FUNCTION_BLOCK HOME_RUN_SEQ
VAR_IN_OUT
	xExecute:		BOOL;
END_VAR
VAR_OUTPUT
	xDone:			BOOL;
END_VAR
VAR
	tpReset:			TP;
	rtDone:				R_TRIG;
	rtExecute:			R_TRIG;
	ftTimePulse:		F_TRIG;
	tpTimePulse:		TP;
	lrTargetPos:		LREAL;
	xTransCondition:	BOOL;	
	xTransRelease:		BOOL;
	SFCInit:			BOOL;
	SFCReset:			BOOL;	
	SFCError:			BOOL;
END_VAR

rtDone(CLK:=xDone);
IF rtDone.Q THEN
	xTransRelease:=FALSE;	
	SFCReset:=TRUE;
END_IF

rtExecute(CLK:=xExecute);
IF rtExecute.Q THEN
	xTransRelease:=TRUE;
	SFCReset:=FALSE;
END_IF

IF xExecute THEN
	aSEQ_ACT();
END_IF

tpReset(IN:=SFCError, PT:=T#250MS);
SFCReset:= tpReset.Q;

ACTION ACK_DONE_AXIS_active:
IF G_sAxisDone.X OR G_sAxisDone.Y OR G_sAxisDone.Z OR G_sAxisDone.c THEN
	G_sAckAxisDone.X:=TRUE;
	G_sAckAxisDone.Y:=TRUE;
	G_sAckAxisDone.Z:=TRUE;
	G_sAckAxisDone.C:=TRUE;
ELSE
	G_sAckAxisDone.X:=FALSE;
	G_sAckAxisDone.Y:=FALSE;
	G_sAckAxisDone.Z:=FALSE;
	G_sAckAxisDone.C:=FALSE;
END_IF

xTransCondition:= NOT G_sAckAxisDone.X AND NOT G_sAckAxisDone.Y AND NOT G_sAckAxisDone.Z AND NOT G_sAckAxisDone.C;
END_ACTION

ACTION aSEQ_ACT:
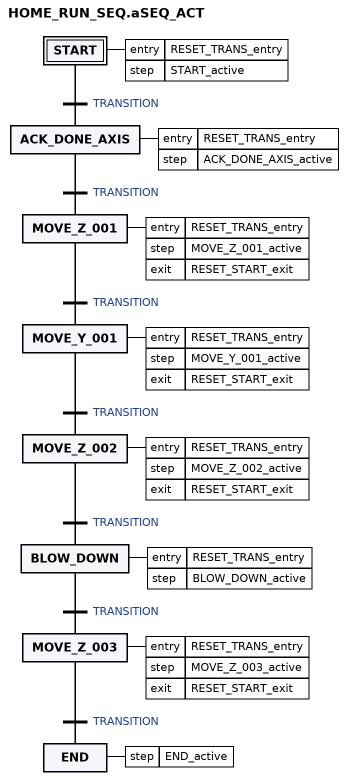
INITIAL_STEP START:
    RESET_TRANS_entry(P1);  // entry action
    START_active(N);  // step action
END_STEP
TRANSITION FROM START TO ACK_DONE_AXIS
    := TRANSITION;
END_TRANSITION
STEP ACK_DONE_AXIS:
    RESET_TRANS_entry(P1);  // entry action
    ACK_DONE_AXIS_active(N);  // step action
END_STEP
TRANSITION FROM ACK_DONE_AXIS TO MOVE_Z_001
    := TRANSITION;
END_TRANSITION
STEP MOVE_Z_001:
    RESET_TRANS_entry(P1);  // entry action
    MOVE_Z_001_active(N);  // step action
    RESET_START_exit(P0);  // exit action
END_STEP
TRANSITION FROM MOVE_Z_001 TO MOVE_Y_001
    := TRANSITION;
END_TRANSITION
STEP MOVE_Y_001:
    RESET_TRANS_entry(P1);  // entry action
    MOVE_Y_001_active(N);  // step action
    RESET_START_exit(P0);  // exit action
END_STEP
TRANSITION FROM MOVE_Y_001 TO MOVE_Z_002
    := TRANSITION;
END_TRANSITION
STEP MOVE_Z_002:
    RESET_TRANS_entry(P1);  // entry action
    MOVE_Z_002_active(N);  // step action
    RESET_START_exit(P0);  // exit action
END_STEP
TRANSITION FROM MOVE_Z_002 TO BLOW_DOWN
    := TRANSITION;
END_TRANSITION
STEP BLOW_DOWN:
    RESET_TRANS_entry(P1);  // entry action
    BLOW_DOWN_active(N);  // step action
END_STEP
TRANSITION FROM BLOW_DOWN TO MOVE_Z_003
    := TRANSITION;
END_TRANSITION
STEP MOVE_Z_003:
    RESET_TRANS_entry(P1);  // entry action
    MOVE_Z_003_active(N);  // step action
    RESET_START_exit(P0);  // exit action
END_STEP
TRANSITION FROM MOVE_Z_003 TO END
    := TRANSITION;
END_TRANSITION
STEP END:
    END_active(N);  // step action
END_STEP
END_ACTION

ACTION BLOW_DOWN_active:
tpTimePulse(IN:=NOT tpTimePulse.Q, PT:=T#3000MS);
ftTimePulse(CLK:=tpTimePulse.Q);
xTransCondition:= ftTimePulse.Q;
END_ACTION

ACTION END_active:
xDone:=TRUE;
xTransCondition:=FALSE;
END_ACTION

ACTION MOVE_Y_001_active:
G_sTargetPosition.Y:= G_asIndividualAxisPositions[CE_AXIS_Y].Positions[1].Target;
G_sStartToPos.Y:= TRUE;

xTransCondition:= G_sAxisDone.Y;
END_ACTION

ACTION MOVE_Z_001_active:
G_sTargetPosition.Z:= G_asIndividualAxisPositions[CE_AXIS_Z].Positions[1].Target;
G_sStartToPos.Z:= TRUE;

xTransCondition:= G_sAxisDone.Z;
END_ACTION

ACTION MOVE_Z_002_active:
G_sTargetPosition.Z:= G_asIndividualAxisPositions[CE_AXIS_Z].Positions[2].Target;
G_sStartToPos.Z:= TRUE;

xTransCondition:= G_sAxisDone.Z;
END_ACTION

ACTION MOVE_Z_003_active:
G_sTargetPosition.Z:= G_asIndividualAxisPositions[CE_AXIS_Z].Positions[1].Target;
G_sStartToPos.Z:= TRUE;

xTransCondition:= G_sAxisDone.Z;
END_ACTION

ACTION RESET_START_exit:
IF G_sAxisDone.X OR G_sAxisDone.Y OR G_sAxisDone.Z OR G_sAxisDone.c THEN
	G_sAckAxisDone.X:=TRUE;
	G_sAckAxisDone.Y:=TRUE;
	G_sAckAxisDone.Z:=TRUE;
	G_sAckAxisDone.C:=TRUE;
ELSE
	G_sAckAxisDone.X:=FALSE;
	G_sAckAxisDone.Y:=FALSE;
	G_sAckAxisDone.Z:=FALSE;
	G_sAckAxisDone.C:=FALSE;
	
	G_sStartToPos.X:=FALSE;
	G_sStartToPos.Y:=FALSE;
	G_sStartToPos.Z:=FALSE;
	G_sStartToPos.C:=FALSE;
END_IF
END_ACTION

ACTION RESET_TRANS_entry:
xTransCondition:= false;
END_ACTION

ACTION START_active:
xDone:=FALSE;
xTransCondition:= NOT xDone;
END_ACTION

TRANSITION TRANSITION:
xTransRelease AND xTransCondition
END_TRANSITION

END_FUNCTION_BLOCK

(* stored: Version 1.1.0.1, ProductVersion 3.1.4022.18
   POU HOME_RUN_SEQ: Id {f74819b4-46ed-48b4-aaf7-d3e507270c38}, SpecialFunc None
   Folder xActive: Id {b1ce9070-77e4-478c-8b3c-0dd9542fd3b0}
   Folder xEntry: Id {045399df-d91f-44e4-9ff5-7400a788c9a3}
   Folder xExit: Id {3b834dd8-5bbb-46dd-9ef0-384de5e2a6b1}
   Folder xTrans: Id {b1dccb1a-ca2a-4f92-ab7f-da8fb147bdbf}
   Action ACK_DONE_AXIS_active: Id {ca99672c-aadc-4547-bdce-dfdeec11da57}
   Action aSEQ_ACT: Id {a8a3a2e5-6a7c-4f33-ae32-7e4e1df91ecc}
   Action BLOW_DOWN_active: Id {8a29b316-4871-44bd-9b82-38cc7d634cfb}
   Action END_active: Id {96baccb2-656f-4685-8ab9-25314354e412}
   Action MOVE_Y_001_active: Id {1eba28ff-16a2-4bd0-8a89-f6185b3d576a}
   Action MOVE_Z_001_active: Id {2e66abb4-1854-4be0-bba0-d2ebdce71273}
   Action MOVE_Z_002_active: Id {7866d3e2-53f6-4d20-9b98-f04168b57650}
   Action MOVE_Z_003_active: Id {0399ee95-11c6-416c-b740-e93d8b6bf0e1}
   Action RESET_START_exit: Id {e7ad9f97-485d-46f7-9a5d-d0db20fad6f0}
   Action RESET_TRANS_entry: Id {05a54e68-4169-42e1-a689-ec647c0e02e5}
   Action START_active: Id {59536f3b-c21b-4d29-8d76-e9dd1d163e96}
   Transition TRANSITION: Id {6418d888-ac6f-45c7-82cd-4b4b88ab0958} *)
